// TIA Portal V19 export
ORGANIZATION_BLOCK "Main"   // OB1, LAD, ProgramCycle
TITLE = "Main Program Sweep (Cycle)"
{ S7_Optimized_Access := 'TRUE' }
// stored: SetENOAutomatically false
   VAR_INPUT
      Initial_Call : Bool;   // Initial call of this OB
      Remanence : Bool;   // =True, if remanent data are available
   END_VAR
   VAR_TEMP   // added for the SCL form of the ladder/FBD networks
      _w1 : Bool;
   END_VAR
BEGIN

REGION Network 1
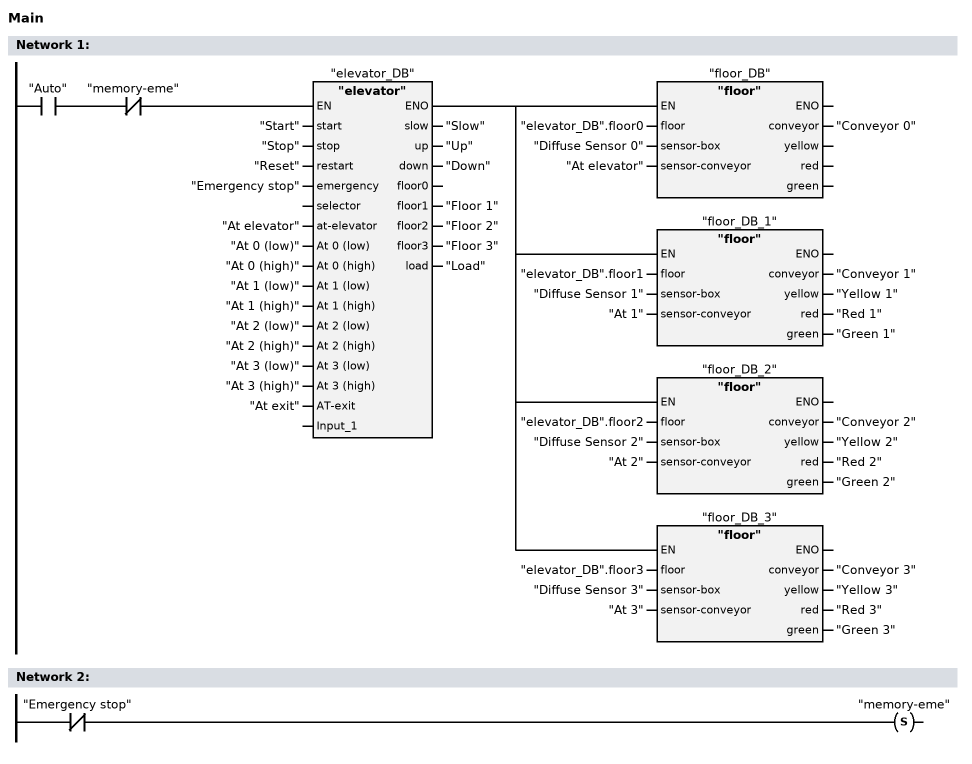
   RUNG wire#powerrail
      Contact( "Auto" )
      I_Contact( "memory-eme" )
      "elevator_DB"(start := "Start", stop := "Stop", restart := "Reset", emergency := "Emergency stop", selector :=, "at-elevator" := "At elevator", "At 0 (low)" := "At 0 (low)", "At 0 (high)" := "At 0 (high)", "At 1 (low)" := "At 1 (low)", "At 1 (high)" := "At 1 (high)", "At 2 (low)" := "At 2 (low)", "At 2 (high)" := "At 2 (high)", "At 3 (low)" := "At 3 (low)", "At 3 (high)" := "At 3 (high)", "AT-exit" := "At exit", Input_1 :=, slow => "Slow", up => "Up", down => "Down", floor0 =>, floor1 => "Floor 1", floor2 => "Floor 2", floor3 => "Floor 3", load => "Load")
      wire#w1
      "floor_DB"(floor := "elevator_DB".floor0, "sensor-box" := "Diffuse Sensor 0", "sensor-conveyor" := "At elevator", conveyor => "Conveyor 0", yellow =>, red =>, green =>)
   END_RUNG
   RUNG wire#w1
      "floor_DB_1"(floor := "elevator_DB".floor1, "sensor-box" := "Diffuse Sensor 1", "sensor-conveyor" := "At 1", conveyor => "Conveyor 1", yellow => "Yellow 1", red => "Red 1", green => "Green 1")
   END_RUNG
   RUNG wire#w1
      "floor_DB_2"(floor := "elevator_DB".floor2, "sensor-box" := "Diffuse Sensor 2", "sensor-conveyor" := "At 2", conveyor => "Conveyor 2", yellow => "Yellow 2", red => "Red 2", green => "Green 2")
   END_RUNG
   RUNG wire#w1
      "floor_DB_3"(floor := "elevator_DB".floor3, "sensor-box" := "Diffuse Sensor 3", "sensor-conveyor" := "At 3", conveyor => "Conveyor 3", yellow => "Yellow 3", red => "Red 3", green => "Green 3")
   END_RUNG
   // the same network as SCL:
   "elevator_DB"(EN := "Auto" AND NOT "memory-eme",   // "elevator"
                 start := "Start",
                 stop := "Stop",
                 restart := "Reset",
                 emergency := "Emergency stop",
                 "at-elevator" := "At elevator",
                 "At 0 (low)" := "At 0 (low)",
                 "At 0 (high)" := "At 0 (high)",
                 "At 1 (low)" := "At 1 (low)",
                 "At 1 (high)" := "At 1 (high)",
                 "At 2 (low)" := "At 2 (low)",
                 "At 2 (high)" := "At 2 (high)",
                 "At 3 (low)" := "At 3 (low)",
                 "At 3 (high)" := "At 3 (high)",
                 "AT-exit" := "At exit",
                 slow => "Slow",
                 up => "Up",
                 down => "Down",
                 floor1 => "Floor 1",
                 floor2 => "Floor 2",
                 floor3 => "Floor 3",
                 load => "Load",
                 ENO => #_w1);
   IF #_w1 THEN
       "floor_DB"(floor := "elevator_DB".floor0,   // "floor"
                  "sensor-box" := "Diffuse Sensor 0",
                  "sensor-conveyor" := "At elevator",
                  conveyor => "Conveyor 0");
       "floor_DB_1"(floor := "elevator_DB".floor1,   // "floor"
                    "sensor-box" := "Diffuse Sensor 1",
                    "sensor-conveyor" := "At 1",
                    conveyor => "Conveyor 1",
                    yellow => "Yellow 1",
                    red => "Red 1",
                    green => "Green 1");
       "floor_DB_2"(floor := "elevator_DB".floor2,   // "floor"
                    "sensor-box" := "Diffuse Sensor 2",
                    "sensor-conveyor" := "At 2",
                    conveyor => "Conveyor 2",
                    yellow => "Yellow 2",
                    red => "Red 2",
                    green => "Green 2");
       "floor_DB_3"(floor := "elevator_DB".floor3,   // "floor"
                    "sensor-box" := "Diffuse Sensor 3",
                    "sensor-conveyor" := "At 3",
                    conveyor => "Conveyor 3",
                    yellow => "Yellow 3",
                    red => "Red 3",
                    green => "Green 3");
   END_IF;
END_REGION

REGION Network 2
   RUNG wire#powerrail
      I_Contact( "Emergency stop" )
      S_Coil( "memory-eme" )
   END_RUNG
   // the same network as SCL:
   IF NOT "Emergency stop" THEN "memory-eme" := TRUE; END_IF;
END_REGION
END_ORGANIZATION_BLOCK
